(*			
	RafalOS
	Rafał Osajda		20.11.2025		TC 4024.66
	Moduł przygotowania danych dla Okna głównego w trybie ręcznym
*)
FUNCTION_BLOCK FB_MCHMIPrepareDataForScreen_00_03 EXTENDS FB_MCHMIPrepareDataForScreen IMPLEMENTS ITF_MCHMIPrepareDataForScreen
VAR
	itfMachineControlHMI	: ITF_MCHMIMachineControl_HMI_PrepScr_00_03;
	refstData				: REFERENCE TO ST_MCHMIPrepareScreen_00_03;
END_VAR

(*			
	RafalOS
	Rafał Osajda		19.11.2025		TC 4024.66
	Czyści danych przy zmienia ramki po poprzedniej ramce
*)
METHOD PUBLIC ClearAfterScreen : BOOL
VAR_INPUT
END_VAR
SUPER^.ClearAfterScreen ();
END_METHOD

METHOD PUBLIC LinkDataHMI_00_03 : BOOL
VAR_INPUT
	refstData				: REFERENCE TO ST_MCHMIPrepareScreen_00_03;
END_VAR
THIS^.refstData REF= refstData;
END_METHOD

METHOD PUBLIC LinkMachineControlHMI : BOOL
VAR_INPUT
	fbMachineControlHMI	: ITF_MCHMIMachineControl_HMI_PrepScr_00_03;
END_VAR
this^.itfMachineControlHMI := fbMachineControlHMI;
END_METHOD

(*			
	RafalOS
	Rafał Osajda		14.11.2025		TC 4024.66
	Metoda przygotowywania danych dla HMI 
	W niej odbywa się odpytywanie właściego elementu przez łącznik
*)
METHOD PUBLIC PrepareDataForHMI : BOOL
VAR_INPUT
END_VAR
SUPER^.PrepareDataForHMI ();
END_METHOD

(*			
	RafalOS
	Rafał Osajda		19.11.2025		TC 4024.66
	Przygotowanie ramki pood tamke do wyświetlenia - tylko przygotowanie a nie przygotowanie danych do wyświetlenia
*)
METHOD PUBLIC PrepareForScreen : BOOL
VAR_INPUT
END_VAR
SUPER^.PrepareForScreen ();
END_METHOD

END_FUNCTION_BLOCK

(* stored: Version 1.1.0.1
   POU FB_MCHMIPrepareDataForScreen_00_03: Id {61612011-d71e-0c9a-0d06-8a18be7896f8}, SpecialFunc None
   Folder ITF_PDFS: Id {79bb0956-62e1-0fa6-1279-767cec79fe6e}
   Method ClearAfterScreen: Id {fac2fefe-2c63-0cb8-22fb-1cc13e2844fd}
   Method LinkDataHMI_00_03: Id {b88ce0fa-5a2b-005b-19f5-155154026cfd}
   Method LinkMachineControlHMI: Id {3b562800-86e2-089a-2f00-940d5f6fd1c7}
   Method PrepareDataForHMI: Id {983810b3-ef02-0f4c-0cd0-95893af2cdfd}
   Method PrepareForScreen: Id {9631ae1b-8962-0936-3afe-26e0b4842463} *)
